{attribute addProperty BoxType "EP7402-0057-0017"}
{attribute addProperty Id "Ready_to_enableBIT10.1251ReadyBIT10.1252WarningBIT10.1253ErrorBIT10.1254Moving_positiveBIT10.1255Moving_negativeBIT10.1256TxPDO_ToggleBIT10.12516"}
{attribute addProperty CRC "650857170"}
{attribute addProperty SizeInBites "16"}
{attribute addProperty SizeInBytes "2"}
TYPE Status_26CB4AD2 :
STRUCT
	{attribute addProperty Name "Ready_to_enable"}
	Ready_to_enable : BIT;
	{attribute addProperty Name "Ready"}
	Ready : BIT;
	{attribute addProperty Name "Warning"}
	Warning : BIT;
	{attribute addProperty Name "Error"}
	Error : BIT;
	{attribute addProperty Name "Moving_positive"}
	Moving_positive : BIT;
	{attribute addProperty Name "Moving_negative"}
	Moving_negative : BIT;
	{attribute 'hide'}
	reserve_1_BIT_0 : BIT;
	{attribute 'hide'}
	reserve_1_BIT_1 : BIT;
	{attribute 'hide'}
	reserve_1_BIT_2 : BIT;
	{attribute 'hide'}
	reserve_1_BIT_3 : BIT;
	{attribute 'hide'}
	reserve_1_BIT_4 : BIT;
	{attribute 'hide'}
	reserve_1_BIT_5 : BIT;
	{attribute 'hide'}
	reserve_1_BIT_6 : BIT;
	{attribute 'hide'}
	reserve_1_BIT_7 : BIT;
	{attribute 'hide'}
	reserve_1_BIT_8 : BIT;
	{attribute addProperty Name "TxPDO_Toggle"}
	TxPDO_Toggle : BIT;
END_STRUCT
END_TYPE

(* stored: Version 1.2.0.0, ProductVersion 3.1.4024.9
   DUT Status_26CB4AD2: Id {8688e98e-557e-4a91-92d4-76a026d233ea} *)
